TYPE FB_ServoAchse_Cmd :
STRUCT
	enable 			: BOOL;
	disable			: BOOL;
	hand			: FB_ServoAchse_Hand;
	fahreAbs		: BOOL;
	position		: LREAL;
	geschwindigkeit	: LREAL;
	halt			: BOOL;
	reset 			: BOOL;
END_STRUCT
END_TYPE

(* stored: Version 1.1.0.1, ProductVersion 3.1.4018.5
   DUT FB_ServoAchse_Cmd: Id {283a869b-65f9-4f42-b638-ee290c316174} *)
